// TIA Portal V20 export
ORGANIZATION_BLOCK "Startup"   // OB100, LAD, Startup
TITLE = "Complete Restart"
// stored: AutoNumber false, IsIECCheckEnabled true, SetENOAutomatically true
   VAR_INPUT
      LostRetentive : Bool;   // True if retentive data are lost
      LostRTC : Bool;   // True if date and time are lost
   END_VAR
   VAR_TEMP
      tempError : Bool;
      tempStatus : Word;
      tempDiagnostics : "LAF_typeDiagnosticsSimple";
   END_VAR
BEGIN

REGION Network 1: Erster Zyklus bit setzen / Set first cycle bit
   // Setze das "erster Zyklus" Signal und die Signale immer EIN sowie immer AUS / Set the first cycle signal
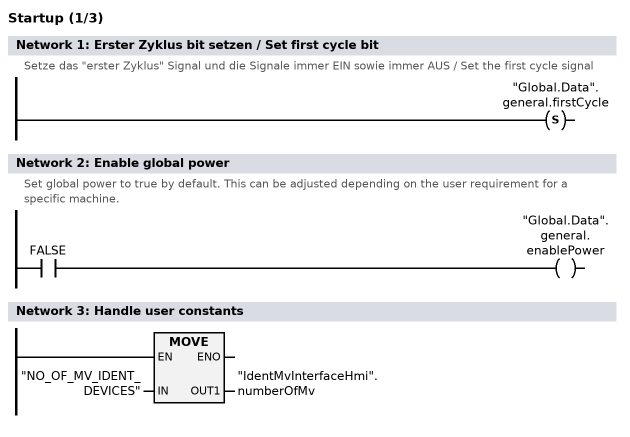
   RUNG wire#powerrail
      S_Coil( "Global.Data".general.firstCycle )
   END_RUNG
   // the same network as SCL:
   "Global.Data".general.firstCycle := TRUE;
END_REGION

REGION Network 2: Enable global power
   // Set global power to true by default. This can be adjusted depending on the user requirement for a specific machine.
   RUNG wire#powerrail
      Contact( FALSE )
      Coil( "Global.Data".general.enablePower )
   END_RUNG
   // the same network as SCL:
   "Global.Data".general.enablePower := FALSE;
END_REGION

REGION Network 3: Handle user constants
   RUNG wire#powerrail
      Move(in := "NO_OF_MV_IDENT_DEVICES", out1 => "IdentMvInterfaceHmi".numberOfMv)
   END_RUNG
   // the same network as SCL:
   "IdentMvInterfaceHmi".numberOfMv := "NO_OF_MV_IDENT_DEVICES";
END_REGION

REGION Network 4: Set drive objects for drive diagnostic
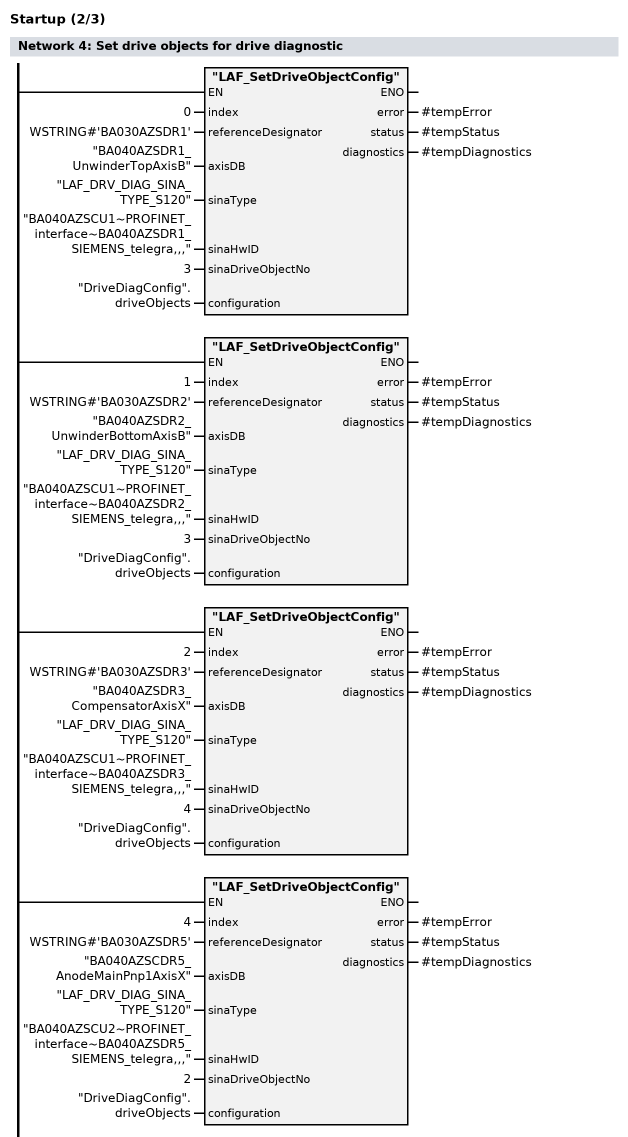
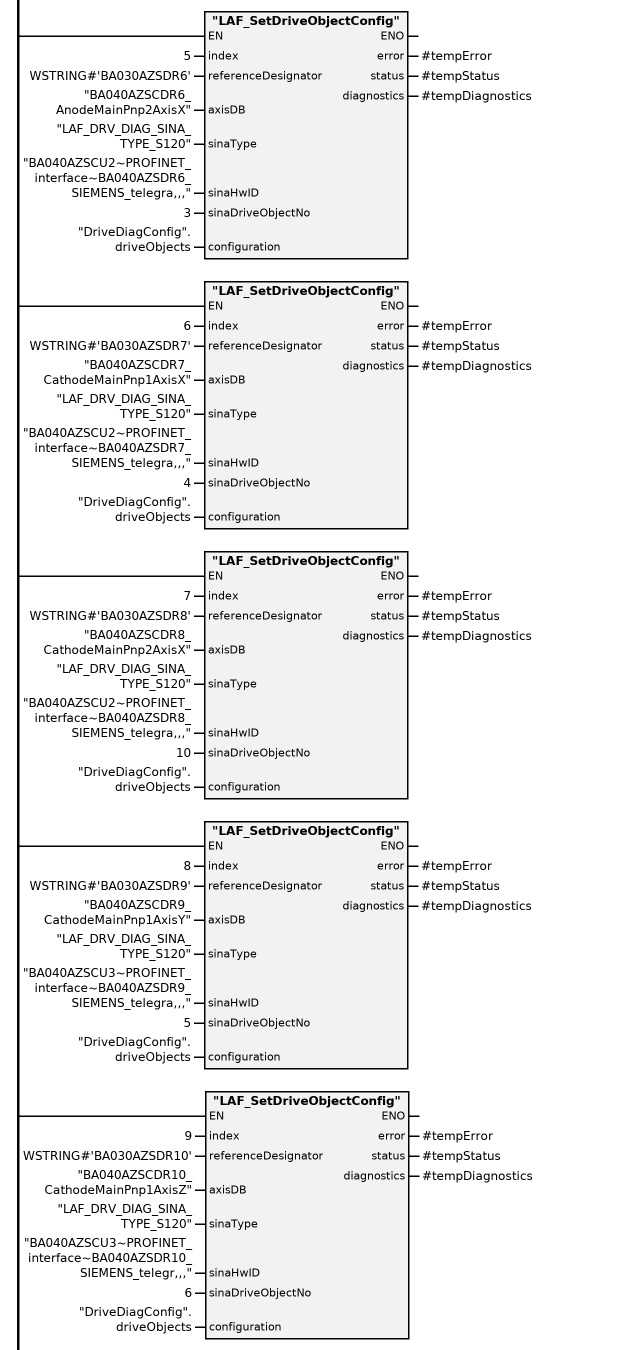
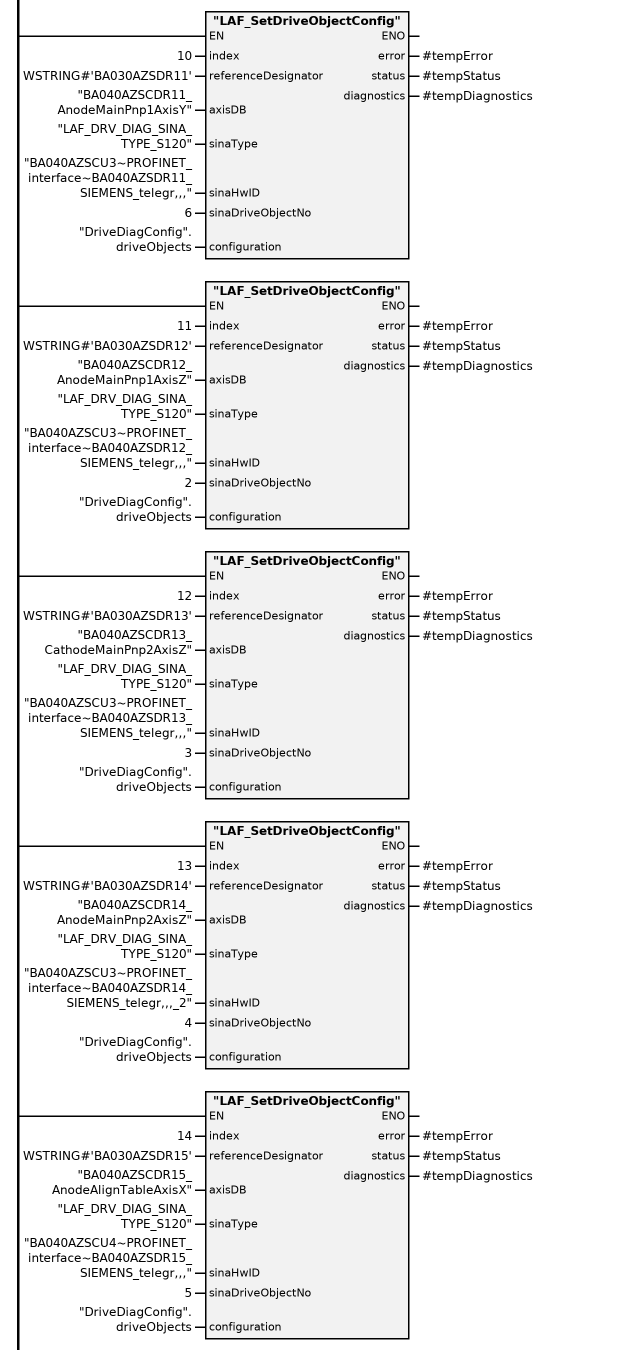
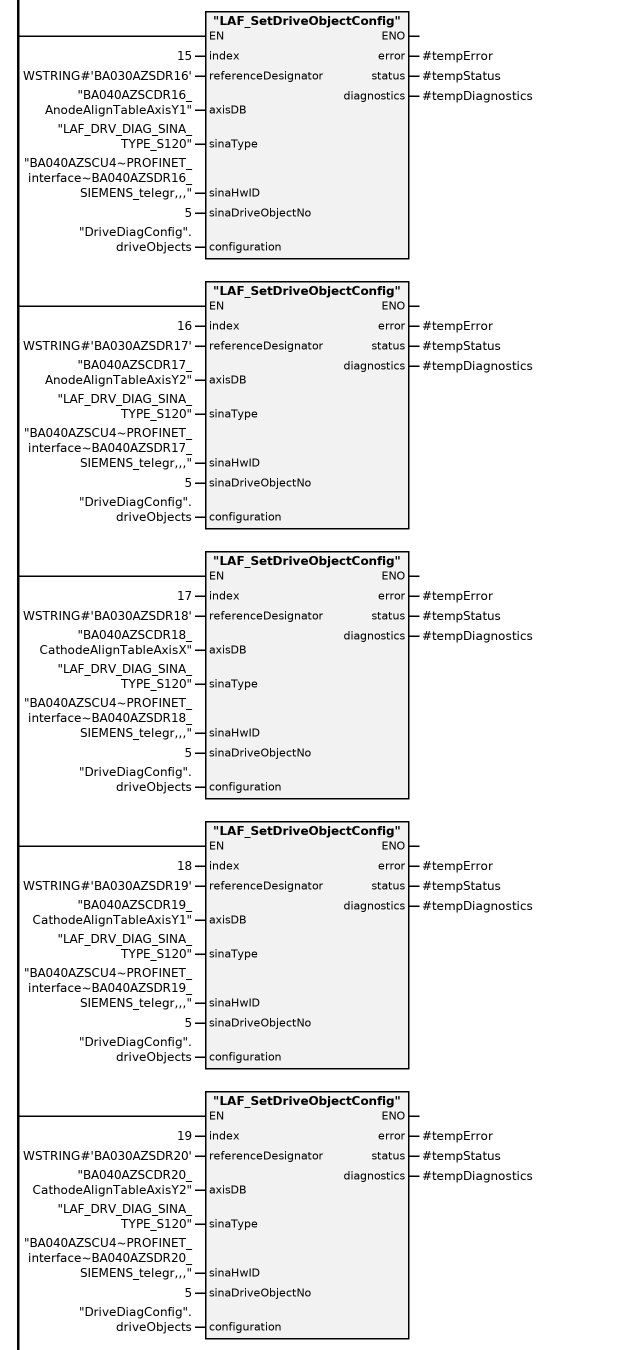
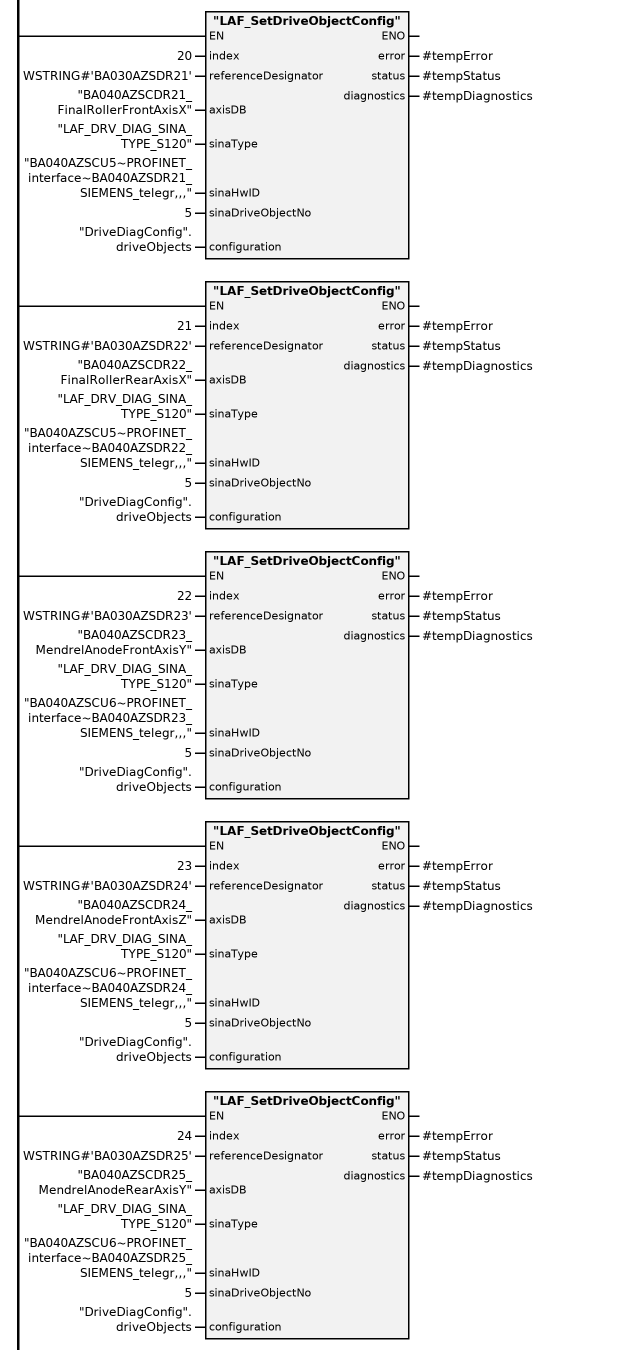
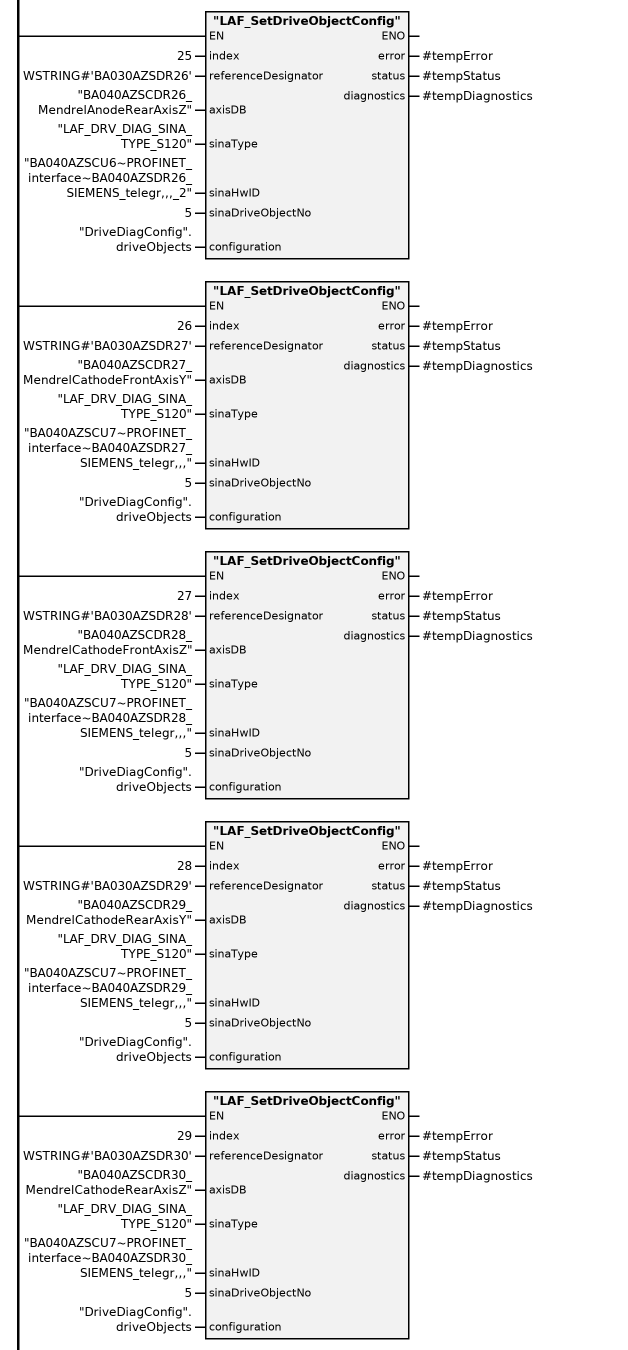
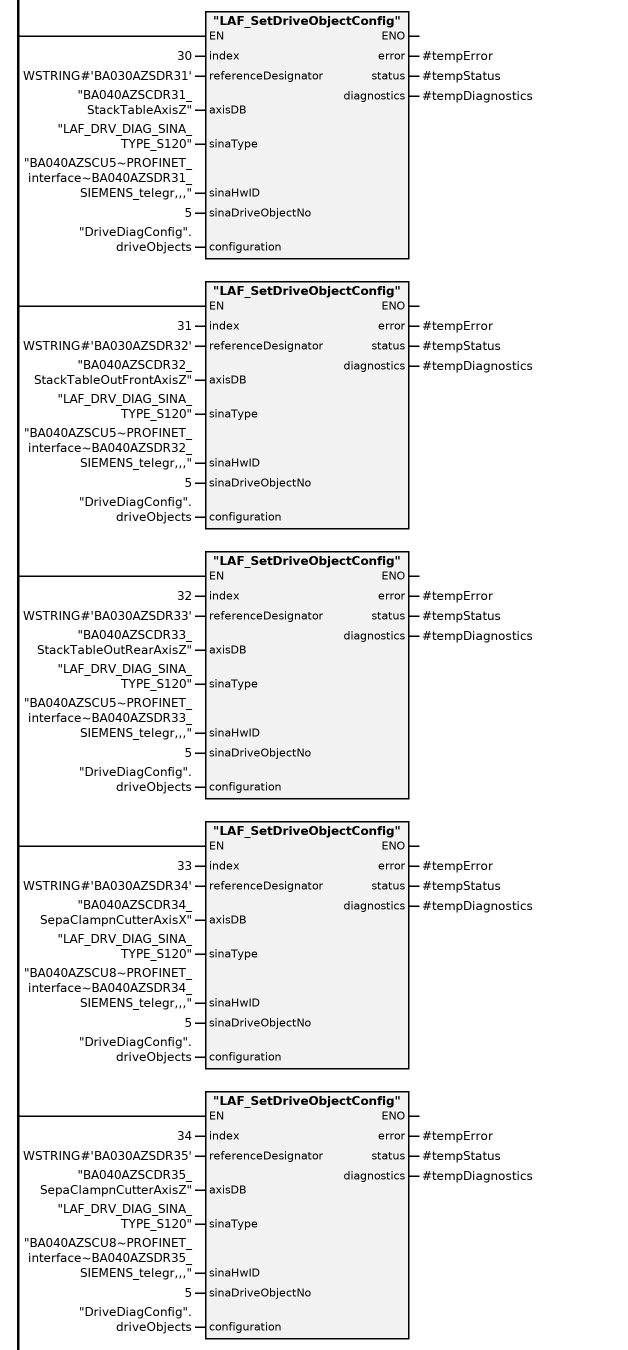
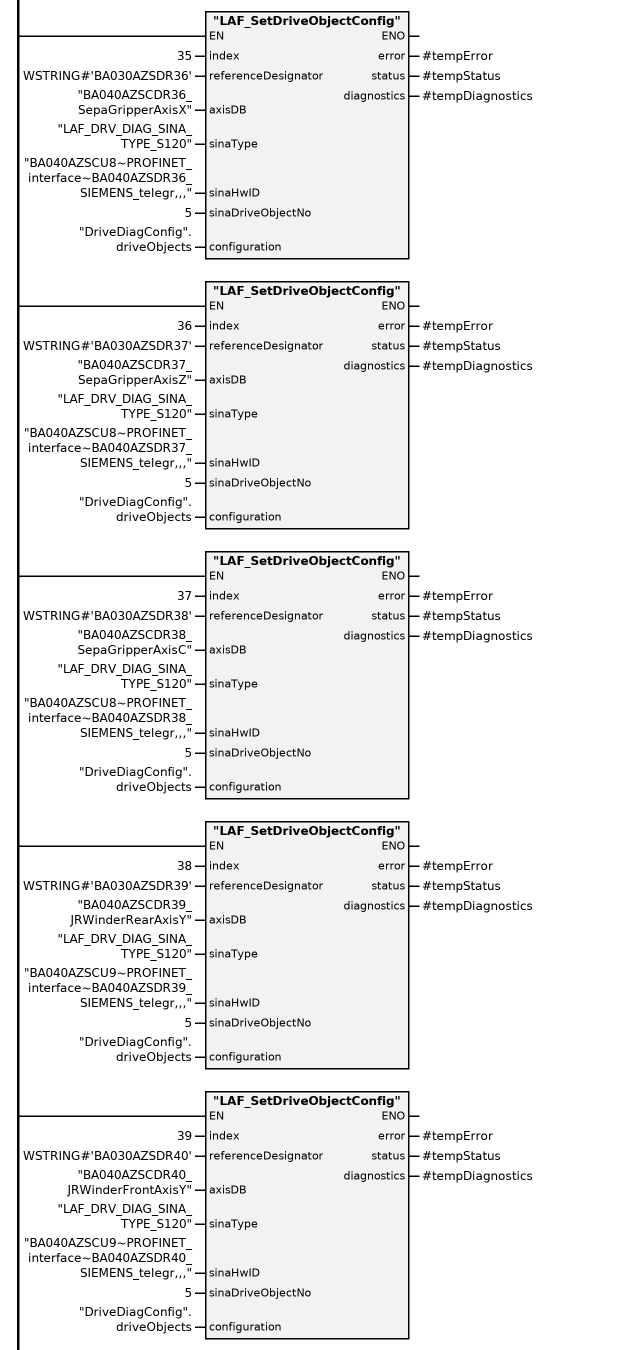
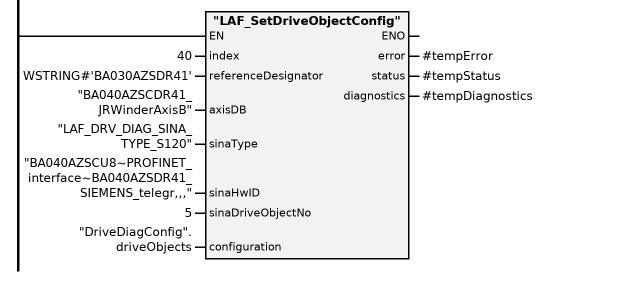
   RUNG wire#powerrail
      "LAF_SetDriveObjectConfig"(index := 0, referenceDesignator := WSTRING#'BA030AZSDR1', axisDB := "BA040AZSDR1_UnwinderTopAxisB", sinaType := "LAF_DRV_DIAG_SINA_TYPE_S120", sinaHwID := "BA040AZSCU1~PROFINET_interface~BA040AZSDR1_SIEMENS_telegra,,,", sinaDriveObjectNo := 3, configuration := "DriveDiagConfig".driveObjects, error => #tempError, status => #tempStatus, diagnostics => #tempDiagnostics)
   END_RUNG
   RUNG wire#powerrail
      "LAF_SetDriveObjectConfig"(index := 1, referenceDesignator := WSTRING#'BA030AZSDR2', axisDB := "BA040AZSDR2_UnwinderBottomAxisB", sinaType := "LAF_DRV_DIAG_SINA_TYPE_S120", sinaHwID := "BA040AZSCU1~PROFINET_interface~BA040AZSDR2_SIEMENS_telegra,,,", sinaDriveObjectNo := 3, configuration := "DriveDiagConfig".driveObjects, error => #tempError, status => #tempStatus, diagnostics => #tempDiagnostics)
   END_RUNG
   RUNG wire#powerrail
      "LAF_SetDriveObjectConfig"(index := 2, referenceDesignator := WSTRING#'BA030AZSDR3', axisDB := "BA040AZSDR3_CompensatorAxisX", sinaType := "LAF_DRV_DIAG_SINA_TYPE_S120", sinaHwID := "BA040AZSCU1~PROFINET_interface~BA040AZSDR3_SIEMENS_telegra,,,", sinaDriveObjectNo := 4, configuration := "DriveDiagConfig".driveObjects, error => #tempError, status => #tempStatus, diagnostics => #tempDiagnostics)
   END_RUNG
   RUNG wire#powerrail
      "LAF_SetDriveObjectConfig"(index := 4, referenceDesignator := WSTRING#'BA030AZSDR5', axisDB := "BA040AZSCDR5_AnodeMainPnp1AxisX", sinaType := "LAF_DRV_DIAG_SINA_TYPE_S120", sinaHwID := "BA040AZSCU2~PROFINET_interface~BA040AZSDR5_SIEMENS_telegra,,,", sinaDriveObjectNo := 2, configuration := "DriveDiagConfig".driveObjects, error => #tempError, status => #tempStatus, diagnostics => #tempDiagnostics)
   END_RUNG
   RUNG wire#powerrail
      "LAF_SetDriveObjectConfig"(index := 5, referenceDesignator := WSTRING#'BA030AZSDR6', axisDB := "BA040AZSCDR6_AnodeMainPnp2AxisX", sinaType := "LAF_DRV_DIAG_SINA_TYPE_S120", sinaHwID := "BA040AZSCU2~PROFINET_interface~BA040AZSDR6_SIEMENS_telegra,,,", sinaDriveObjectNo := 3, configuration := "DriveDiagConfig".driveObjects, error => #tempError, status => #tempStatus, diagnostics => #tempDiagnostics)
   END_RUNG
   RUNG wire#powerrail
      "LAF_SetDriveObjectConfig"(index := 6, referenceDesignator := WSTRING#'BA030AZSDR7', axisDB := "BA040AZSCDR7_CathodeMainPnp1AxisX", sinaType := "LAF_DRV_DIAG_SINA_TYPE_S120", sinaHwID := "BA040AZSCU2~PROFINET_interface~BA040AZSDR7_SIEMENS_telegra,,,", sinaDriveObjectNo := 4, configuration := "DriveDiagConfig".driveObjects, error => #tempError, status => #tempStatus, diagnostics => #tempDiagnostics)
   END_RUNG
   RUNG wire#powerrail
      "LAF_SetDriveObjectConfig"(index := 7, referenceDesignator := WSTRING#'BA030AZSDR8', axisDB := "BA040AZSCDR8_CathodeMainPnp2AxisX", sinaType := "LAF_DRV_DIAG_SINA_TYPE_S120", sinaHwID := "BA040AZSCU2~PROFINET_interface~BA040AZSDR8_SIEMENS_telegra,,,", sinaDriveObjectNo := 10, configuration := "DriveDiagConfig".driveObjects, error => #tempError, status => #tempStatus, diagnostics => #tempDiagnostics)
   END_RUNG
   RUNG wire#powerrail
      "LAF_SetDriveObjectConfig"(index := 8, referenceDesignator := WSTRING#'BA030AZSDR9', axisDB := "BA040AZSCDR9_CathodeMainPnp1AxisY", sinaType := "LAF_DRV_DIAG_SINA_TYPE_S120", sinaHwID := "BA040AZSCU3~PROFINET_interface~BA040AZSDR9_SIEMENS_telegra,,,", sinaDriveObjectNo := 5, configuration := "DriveDiagConfig".driveObjects, error => #tempError, status => #tempStatus, diagnostics => #tempDiagnostics)
   END_RUNG
   RUNG wire#powerrail
      "LAF_SetDriveObjectConfig"(index := 9, referenceDesignator := WSTRING#'BA030AZSDR10', axisDB := "BA040AZSCDR10_CathodeMainPnp1AxisZ", sinaType := "LAF_DRV_DIAG_SINA_TYPE_S120", sinaHwID := "BA040AZSCU3~PROFINET_interface~BA040AZSDR10_SIEMENS_telegr,,,", sinaDriveObjectNo := 6, configuration := "DriveDiagConfig".driveObjects, error => #tempError, status => #tempStatus, diagnostics => #tempDiagnostics)
   END_RUNG
   RUNG wire#powerrail
      "LAF_SetDriveObjectConfig"(index := 10, referenceDesignator := WSTRING#'BA030AZSDR11', axisDB := "BA040AZSCDR11_AnodeMainPnp1AxisY", sinaType := "LAF_DRV_DIAG_SINA_TYPE_S120", sinaHwID := "BA040AZSCU3~PROFINET_interface~BA040AZSDR11_SIEMENS_telegr,,,", sinaDriveObjectNo := 6, configuration := "DriveDiagConfig".driveObjects, error => #tempError, status => #tempStatus, diagnostics => #tempDiagnostics)
   END_RUNG
   RUNG wire#powerrail
      "LAF_SetDriveObjectConfig"(index := 11, referenceDesignator := WSTRING#'BA030AZSDR12', axisDB := "BA040AZSCDR12_AnodeMainPnp1AxisZ", sinaType := "LAF_DRV_DIAG_SINA_TYPE_S120", sinaHwID := "BA040AZSCU3~PROFINET_interface~BA040AZSDR12_SIEMENS_telegr,,,", sinaDriveObjectNo := 2, configuration := "DriveDiagConfig".driveObjects, error => #tempError, status => #tempStatus, diagnostics => #tempDiagnostics)
   END_RUNG
   RUNG wire#powerrail
      "LAF_SetDriveObjectConfig"(index := 12, referenceDesignator := WSTRING#'BA030AZSDR13', axisDB := "BA040AZSCDR13_CathodeMainPnp2AxisZ", sinaType := "LAF_DRV_DIAG_SINA_TYPE_S120", sinaHwID := "BA040AZSCU3~PROFINET_interface~BA040AZSDR13_SIEMENS_telegr,,,", sinaDriveObjectNo := 3, configuration := "DriveDiagConfig".driveObjects, error => #tempError, status => #tempStatus, diagnostics => #tempDiagnostics)
   END_RUNG
   RUNG wire#powerrail
      "LAF_SetDriveObjectConfig"(index := 13, referenceDesignator := WSTRING#'BA030AZSDR14', axisDB := "BA040AZSCDR14_AnodeMainPnp2AxisZ", sinaType := "LAF_DRV_DIAG_SINA_TYPE_S120", sinaHwID := "BA040AZSCU3~PROFINET_interface~BA040AZSDR14_SIEMENS_telegr,,,_2", sinaDriveObjectNo := 4, configuration := "DriveDiagConfig".driveObjects, error => #tempError, status => #tempStatus, diagnostics => #tempDiagnostics)
   END_RUNG
   RUNG wire#powerrail
      "LAF_SetDriveObjectConfig"(index := 14, referenceDesignator := WSTRING#'BA030AZSDR15', axisDB := "BA040AZSCDR15_AnodeAlignTableAxisX", sinaType := "LAF_DRV_DIAG_SINA_TYPE_S120", sinaHwID := "BA040AZSCU4~PROFINET_interface~BA040AZSDR15_SIEMENS_telegr,,,", sinaDriveObjectNo := 5, configuration := "DriveDiagConfig".driveObjects, error => #tempError, status => #tempStatus, diagnostics => #tempDiagnostics)
   END_RUNG
   RUNG wire#powerrail
      "LAF_SetDriveObjectConfig"(index := 15, referenceDesignator := WSTRING#'BA030AZSDR16', axisDB := "BA040AZSCDR16_AnodeAlignTableAxisY1", sinaType := "LAF_DRV_DIAG_SINA_TYPE_S120", sinaHwID := "BA040AZSCU4~PROFINET_interface~BA040AZSDR16_SIEMENS_telegr,,,", sinaDriveObjectNo := 5, configuration := "DriveDiagConfig".driveObjects, error => #tempError, status => #tempStatus, diagnostics => #tempDiagnostics)
   END_RUNG
   RUNG wire#powerrail
      "LAF_SetDriveObjectConfig"(index := 16, referenceDesignator := WSTRING#'BA030AZSDR17', axisDB := "BA040AZSCDR17_AnodeAlignTableAxisY2", sinaType := "LAF_DRV_DIAG_SINA_TYPE_S120", sinaHwID := "BA040AZSCU4~PROFINET_interface~BA040AZSDR17_SIEMENS_telegr,,,", sinaDriveObjectNo := 5, configuration := "DriveDiagConfig".driveObjects, error => #tempError, status => #tempStatus, diagnostics => #tempDiagnostics)
   END_RUNG
   RUNG wire#powerrail
      "LAF_SetDriveObjectConfig"(index := 17, referenceDesignator := WSTRING#'BA030AZSDR18', axisDB := "BA040AZSCDR18_CathodeAlignTableAxisX", sinaType := "LAF_DRV_DIAG_SINA_TYPE_S120", sinaHwID := "BA040AZSCU4~PROFINET_interface~BA040AZSDR18_SIEMENS_telegr,,,", sinaDriveObjectNo := 5, configuration := "DriveDiagConfig".driveObjects, error => #tempError, status => #tempStatus, diagnostics => #tempDiagnostics)
   END_RUNG
   RUNG wire#powerrail
      "LAF_SetDriveObjectConfig"(index := 18, referenceDesignator := WSTRING#'BA030AZSDR19', axisDB := "BA040AZSCDR19_CathodeAlignTableAxisY1", sinaType := "LAF_DRV_DIAG_SINA_TYPE_S120", sinaHwID := "BA040AZSCU4~PROFINET_interface~BA040AZSDR19_SIEMENS_telegr,,,", sinaDriveObjectNo := 5, configuration := "DriveDiagConfig".driveObjects, error => #tempError, status => #tempStatus, diagnostics => #tempDiagnostics)
   END_RUNG
   RUNG wire#powerrail
      "LAF_SetDriveObjectConfig"(index := 19, referenceDesignator := WSTRING#'BA030AZSDR20', axisDB := "BA040AZSCDR20_CathodeAlignTableAxisY2", sinaType := "LAF_DRV_DIAG_SINA_TYPE_S120", sinaHwID := "BA040AZSCU4~PROFINET_interface~BA040AZSDR20_SIEMENS_telegr,,,", sinaDriveObjectNo := 5, configuration := "DriveDiagConfig".driveObjects, error => #tempError, status => #tempStatus, diagnostics => #tempDiagnostics)
   END_RUNG
   RUNG wire#powerrail
      "LAF_SetDriveObjectConfig"(index := 20, referenceDesignator := WSTRING#'BA030AZSDR21', axisDB := "BA040AZSCDR21_FinalRollerFrontAxisX", sinaType := "LAF_DRV_DIAG_SINA_TYPE_S120", sinaHwID := "BA040AZSCU5~PROFINET_interface~BA040AZSDR21_SIEMENS_telegr,,,", sinaDriveObjectNo := 5, configuration := "DriveDiagConfig".driveObjects, error => #tempError, status => #tempStatus, diagnostics => #tempDiagnostics)
   END_RUNG
   RUNG wire#powerrail
      "LAF_SetDriveObjectConfig"(index := 21, referenceDesignator := WSTRING#'BA030AZSDR22', axisDB := "BA040AZSCDR22_FinalRollerRearAxisX", sinaType := "LAF_DRV_DIAG_SINA_TYPE_S120", sinaHwID := "BA040AZSCU5~PROFINET_interface~BA040AZSDR22_SIEMENS_telegr,,,", sinaDriveObjectNo := 5, configuration := "DriveDiagConfig".driveObjects, error => #tempError, status => #tempStatus, diagnostics => #tempDiagnostics)
   END_RUNG
   RUNG wire#powerrail
      "LAF_SetDriveObjectConfig"(index := 22, referenceDesignator := WSTRING#'BA030AZSDR23', axisDB := "BA040AZSCDR23_MendrelAnodeFrontAxisY", sinaType := "LAF_DRV_DIAG_SINA_TYPE_S120", sinaHwID := "BA040AZSCU6~PROFINET_interface~BA040AZSDR23_SIEMENS_telegr,,,", sinaDriveObjectNo := 5, configuration := "DriveDiagConfig".driveObjects, error => #tempError, status => #tempStatus, diagnostics => #tempDiagnostics)
   END_RUNG
   RUNG wire#powerrail
      "LAF_SetDriveObjectConfig"(index := 23, referenceDesignator := WSTRING#'BA030AZSDR24', axisDB := "BA040AZSCDR24_MendrelAnodeFrontAxisZ", sinaType := "LAF_DRV_DIAG_SINA_TYPE_S120", sinaHwID := "BA040AZSCU6~PROFINET_interface~BA040AZSDR24_SIEMENS_telegr,,,", sinaDriveObjectNo := 5, configuration := "DriveDiagConfig".driveObjects, error => #tempError, status => #tempStatus, diagnostics => #tempDiagnostics)
   END_RUNG
   RUNG wire#powerrail
      "LAF_SetDriveObjectConfig"(index := 24, referenceDesignator := WSTRING#'BA030AZSDR25', axisDB := "BA040AZSCDR25_MendrelAnodeRearAxisY", sinaType := "LAF_DRV_DIAG_SINA_TYPE_S120", sinaHwID := "BA040AZSCU6~PROFINET_interface~BA040AZSDR25_SIEMENS_telegr,,,", sinaDriveObjectNo := 5, configuration := "DriveDiagConfig".driveObjects, error => #tempError, status => #tempStatus, diagnostics => #tempDiagnostics)
   END_RUNG
   RUNG wire#powerrail
      "LAF_SetDriveObjectConfig"(index := 25, referenceDesignator := WSTRING#'BA030AZSDR26', axisDB := "BA040AZSCDR26_MendrelAnodeRearAxisZ", sinaType := "LAF_DRV_DIAG_SINA_TYPE_S120", sinaHwID := "BA040AZSCU6~PROFINET_interface~BA040AZSDR26_SIEMENS_telegr,,,_2", sinaDriveObjectNo := 5, configuration := "DriveDiagConfig".driveObjects, error => #tempError, status => #tempStatus, diagnostics => #tempDiagnostics)
   END_RUNG
   RUNG wire#powerrail
      "LAF_SetDriveObjectConfig"(index := 26, referenceDesignator := WSTRING#'BA030AZSDR27', axisDB := "BA040AZSCDR27_MendrelCathodeFrontAxisY", sinaType := "LAF_DRV_DIAG_SINA_TYPE_S120", sinaHwID := "BA040AZSCU7~PROFINET_interface~BA040AZSDR27_SIEMENS_telegr,,,", sinaDriveObjectNo := 5, configuration := "DriveDiagConfig".driveObjects, error => #tempError, status => #tempStatus, diagnostics => #tempDiagnostics)
   END_RUNG
   RUNG wire#powerrail
      "LAF_SetDriveObjectConfig"(index := 27, referenceDesignator := WSTRING#'BA030AZSDR28', axisDB := "BA040AZSCDR28_MendrelCathodeFrontAxisZ", sinaType := "LAF_DRV_DIAG_SINA_TYPE_S120", sinaHwID := "BA040AZSCU7~PROFINET_interface~BA040AZSDR28_SIEMENS_telegr,,,", sinaDriveObjectNo := 5, configuration := "DriveDiagConfig".driveObjects, error => #tempError, status => #tempStatus, diagnostics => #tempDiagnostics)
   END_RUNG
   RUNG wire#powerrail
      "LAF_SetDriveObjectConfig"(index := 28, referenceDesignator := WSTRING#'BA030AZSDR29', axisDB := "BA040AZSCDR29_MendrelCathodeRearAxisY", sinaType := "LAF_DRV_DIAG_SINA_TYPE_S120", sinaHwID := "BA040AZSCU7~PROFINET_interface~BA040AZSDR29_SIEMENS_telegr,,,", sinaDriveObjectNo := 5, configuration := "DriveDiagConfig".driveObjects, error => #tempError, status => #tempStatus, diagnostics => #tempDiagnostics)
   END_RUNG
   RUNG wire#powerrail
      "LAF_SetDriveObjectConfig"(index := 29, referenceDesignator := WSTRING#'BA030AZSDR30', axisDB := "BA040AZSCDR30_MendrelCathodeRearAxisZ", sinaType := "LAF_DRV_DIAG_SINA_TYPE_S120", sinaHwID := "BA040AZSCU7~PROFINET_interface~BA040AZSDR30_SIEMENS_telegr,,,", sinaDriveObjectNo := 5, configuration := "DriveDiagConfig".driveObjects, error => #tempError, status => #tempStatus, diagnostics => #tempDiagnostics)
   END_RUNG
   RUNG wire#powerrail
      "LAF_SetDriveObjectConfig"(index := 30, referenceDesignator := WSTRING#'BA030AZSDR31', axisDB := "BA040AZSCDR31_StackTableAxisZ", sinaType := "LAF_DRV_DIAG_SINA_TYPE_S120", sinaHwID := "BA040AZSCU5~PROFINET_interface~BA040AZSDR31_SIEMENS_telegr,,,", sinaDriveObjectNo := 5, configuration := "DriveDiagConfig".driveObjects, error => #tempError, status => #tempStatus, diagnostics => #tempDiagnostics)
   END_RUNG
   RUNG wire#powerrail
      "LAF_SetDriveObjectConfig"(index := 31, referenceDesignator := WSTRING#'BA030AZSDR32', axisDB := "BA040AZSCDR32_StackTableOutFrontAxisZ", sinaType := "LAF_DRV_DIAG_SINA_TYPE_S120", sinaHwID := "BA040AZSCU5~PROFINET_interface~BA040AZSDR32_SIEMENS_telegr,,,", sinaDriveObjectNo := 5, configuration := "DriveDiagConfig".driveObjects, error => #tempError, status => #tempStatus, diagnostics => #tempDiagnostics)
   END_RUNG
   RUNG wire#powerrail
      "LAF_SetDriveObjectConfig"(index := 32, referenceDesignator := WSTRING#'BA030AZSDR33', axisDB := "BA040AZSCDR33_StackTableOutRearAxisZ", sinaType := "LAF_DRV_DIAG_SINA_TYPE_S120", sinaHwID := "BA040AZSCU5~PROFINET_interface~BA040AZSDR33_SIEMENS_telegr,,,", sinaDriveObjectNo := 5, configuration := "DriveDiagConfig".driveObjects, error => #tempError, status => #tempStatus, diagnostics => #tempDiagnostics)
   END_RUNG
   RUNG wire#powerrail
      "LAF_SetDriveObjectConfig"(index := 33, referenceDesignator := WSTRING#'BA030AZSDR34', axisDB := "BA040AZSCDR34_SepaClampnCutterAxisX", sinaType := "LAF_DRV_DIAG_SINA_TYPE_S120", sinaHwID := "BA040AZSCU8~PROFINET_interface~BA040AZSDR34_SIEMENS_telegr,,,", sinaDriveObjectNo := 5, configuration := "DriveDiagConfig".driveObjects, error => #tempError, status => #tempStatus, diagnostics => #tempDiagnostics)
   END_RUNG
   RUNG wire#powerrail
      "LAF_SetDriveObjectConfig"(index := 34, referenceDesignator := WSTRING#'BA030AZSDR35', axisDB := "BA040AZSCDR35_SepaClampnCutterAxisZ", sinaType := "LAF_DRV_DIAG_SINA_TYPE_S120", sinaHwID := "BA040AZSCU8~PROFINET_interface~BA040AZSDR35_SIEMENS_telegr,,,", sinaDriveObjectNo := 5, configuration := "DriveDiagConfig".driveObjects, error => #tempError, status => #tempStatus, diagnostics => #tempDiagnostics)
   END_RUNG
   RUNG wire#powerrail
      "LAF_SetDriveObjectConfig"(index := 35, referenceDesignator := WSTRING#'BA030AZSDR36', axisDB := "BA040AZSCDR36_SepaGripperAxisX", sinaType := "LAF_DRV_DIAG_SINA_TYPE_S120", sinaHwID := "BA040AZSCU8~PROFINET_interface~BA040AZSDR36_SIEMENS_telegr,,,", sinaDriveObjectNo := 5, configuration := "DriveDiagConfig".driveObjects, error => #tempError, status => #tempStatus, diagnostics => #tempDiagnostics)
   END_RUNG
   RUNG wire#powerrail
      "LAF_SetDriveObjectConfig"(index := 36, referenceDesignator := WSTRING#'BA030AZSDR37', axisDB := "BA040AZSCDR37_SepaGripperAxisZ", sinaType := "LAF_DRV_DIAG_SINA_TYPE_S120", sinaHwID := "BA040AZSCU8~PROFINET_interface~BA040AZSDR37_SIEMENS_telegr,,,", sinaDriveObjectNo := 5, configuration := "DriveDiagConfig".driveObjects, error => #tempError, status => #tempStatus, diagnostics => #tempDiagnostics)
   END_RUNG
   RUNG wire#powerrail
      "LAF_SetDriveObjectConfig"(index := 37, referenceDesignator := WSTRING#'BA030AZSDR38', axisDB := "BA040AZSCDR38_SepaGripperAxisC", sinaType := "LAF_DRV_DIAG_SINA_TYPE_S120", sinaHwID := "BA040AZSCU8~PROFINET_interface~BA040AZSDR38_SIEMENS_telegr,,,", sinaDriveObjectNo := 5, configuration := "DriveDiagConfig".driveObjects, error => #tempError, status => #tempStatus, diagnostics => #tempDiagnostics)
   END_RUNG
   RUNG wire#powerrail
      "LAF_SetDriveObjectConfig"(index := 38, referenceDesignator := WSTRING#'BA030AZSDR39', axisDB := "BA040AZSCDR39_JRWinderRearAxisY", sinaType := "LAF_DRV_DIAG_SINA_TYPE_S120", sinaHwID := "BA040AZSCU9~PROFINET_interface~BA040AZSDR39_SIEMENS_telegr,,,", sinaDriveObjectNo := 5, configuration := "DriveDiagConfig".driveObjects, error => #tempError, status => #tempStatus, diagnostics => #tempDiagnostics)
   END_RUNG
   RUNG wire#powerrail
      "LAF_SetDriveObjectConfig"(index := 39, referenceDesignator := WSTRING#'BA030AZSDR40', axisDB := "BA040AZSCDR40_JRWinderFrontAxisY", sinaType := "LAF_DRV_DIAG_SINA_TYPE_S120", sinaHwID := "BA040AZSCU9~PROFINET_interface~BA040AZSDR40_SIEMENS_telegr,,,", sinaDriveObjectNo := 5, configuration := "DriveDiagConfig".driveObjects, error => #tempError, status => #tempStatus, diagnostics => #tempDiagnostics)
   END_RUNG
   RUNG wire#powerrail
      "LAF_SetDriveObjectConfig"(index := 40, referenceDesignator := WSTRING#'BA030AZSDR41', axisDB := "BA040AZSCDR41_JRWinderAxisB", sinaType := "LAF_DRV_DIAG_SINA_TYPE_S120", sinaHwID := "BA040AZSCU8~PROFINET_interface~BA040AZSDR41_SIEMENS_telegr,,,", sinaDriveObjectNo := 5, configuration := "DriveDiagConfig".driveObjects, error => #tempError, status => #tempStatus, diagnostics => #tempDiagnostics)
   END_RUNG
   // the same network as SCL:
   "LAF_SetDriveObjectConfig"(index := 0,
                           referenceDesignator := WSTRING#'BA030AZSDR1',
                           axisDB := "BA040AZSDR1_UnwinderTopAxisB",
                           sinaType := "LAF_DRV_DIAG_SINA_TYPE_S120",
                           sinaHwID := "BA040AZSCU1~PROFINET_interface~BA040AZSDR1_SIEMENS_telegra,,,",
                           sinaDriveObjectNo := 3,
                           configuration := "DriveDiagConfig".driveObjects,
                           error => #tempError,
                           status => #tempStatus,
                           diagnostics => #tempDiagnostics);
   "LAF_SetDriveObjectConfig"(index := 1,
                           referenceDesignator := WSTRING#'BA030AZSDR2',
                           axisDB := "BA040AZSDR2_UnwinderBottomAxisB",
                           sinaType := "LAF_DRV_DIAG_SINA_TYPE_S120",
                           sinaHwID := "BA040AZSCU1~PROFINET_interface~BA040AZSDR2_SIEMENS_telegra,,,",
                           sinaDriveObjectNo := 3,
                           configuration := "DriveDiagConfig".driveObjects,
                           error => #tempError,
                           status => #tempStatus,
                           diagnostics => #tempDiagnostics);
   "LAF_SetDriveObjectConfig"(index := 2,
                           referenceDesignator := WSTRING#'BA030AZSDR3',
                           axisDB := "BA040AZSDR3_CompensatorAxisX",
                           sinaType := "LAF_DRV_DIAG_SINA_TYPE_S120",
                           sinaHwID := "BA040AZSCU1~PROFINET_interface~BA040AZSDR3_SIEMENS_telegra,,,",
                           sinaDriveObjectNo := 4,
                           configuration := "DriveDiagConfig".driveObjects,
                           error => #tempError,
                           status => #tempStatus,
                           diagnostics => #tempDiagnostics);
   "LAF_SetDriveObjectConfig"(index := 4,
                           referenceDesignator := WSTRING#'BA030AZSDR5',
                           axisDB := "BA040AZSCDR5_AnodeMainPnp1AxisX",
                           sinaType := "LAF_DRV_DIAG_SINA_TYPE_S120",
                           sinaHwID := "BA040AZSCU2~PROFINET_interface~BA040AZSDR5_SIEMENS_telegra,,,",
                           sinaDriveObjectNo := 2,
                           configuration := "DriveDiagConfig".driveObjects,
                           error => #tempError,
                           status => #tempStatus,
                           diagnostics => #tempDiagnostics);
   "LAF_SetDriveObjectConfig"(index := 5,
                           referenceDesignator := WSTRING#'BA030AZSDR6',
                           axisDB := "BA040AZSCDR6_AnodeMainPnp2AxisX",
                           sinaType := "LAF_DRV_DIAG_SINA_TYPE_S120",
                           sinaHwID := "BA040AZSCU2~PROFINET_interface~BA040AZSDR6_SIEMENS_telegra,,,",
                           sinaDriveObjectNo := 3,
                           configuration := "DriveDiagConfig".driveObjects,
                           error => #tempError,
                           status => #tempStatus,
                           diagnostics => #tempDiagnostics);
   "LAF_SetDriveObjectConfig"(index := 6,
                           referenceDesignator := WSTRING#'BA030AZSDR7',
                           axisDB := "BA040AZSCDR7_CathodeMainPnp1AxisX",
                           sinaType := "LAF_DRV_DIAG_SINA_TYPE_S120",
                           sinaHwID := "BA040AZSCU2~PROFINET_interface~BA040AZSDR7_SIEMENS_telegra,,,",
                           sinaDriveObjectNo := 4,
                           configuration := "DriveDiagConfig".driveObjects,
                           error => #tempError,
                           status => #tempStatus,
                           diagnostics => #tempDiagnostics);
   "LAF_SetDriveObjectConfig"(index := 7,
                           referenceDesignator := WSTRING#'BA030AZSDR8',
                           axisDB := "BA040AZSCDR8_CathodeMainPnp2AxisX",
                           sinaType := "LAF_DRV_DIAG_SINA_TYPE_S120",
                           sinaHwID := "BA040AZSCU2~PROFINET_interface~BA040AZSDR8_SIEMENS_telegra,,,",
                           sinaDriveObjectNo := 10,
                           configuration := "DriveDiagConfig".driveObjects,
                           error => #tempError,
                           status => #tempStatus,
                           diagnostics => #tempDiagnostics);
   "LAF_SetDriveObjectConfig"(index := 8,
                           referenceDesignator := WSTRING#'BA030AZSDR9',
                           axisDB := "BA040AZSCDR9_CathodeMainPnp1AxisY",
                           sinaType := "LAF_DRV_DIAG_SINA_TYPE_S120",
                           sinaHwID := "BA040AZSCU3~PROFINET_interface~BA040AZSDR9_SIEMENS_telegra,,,",
                           sinaDriveObjectNo := 5,
                           configuration := "DriveDiagConfig".driveObjects,
                           error => #tempError,
                           status => #tempStatus,
                           diagnostics => #tempDiagnostics);
   "LAF_SetDriveObjectConfig"(index := 9,
                           referenceDesignator := WSTRING#'BA030AZSDR10',
                           axisDB := "BA040AZSCDR10_CathodeMainPnp1AxisZ",
                           sinaType := "LAF_DRV_DIAG_SINA_TYPE_S120",
                           sinaHwID := "BA040AZSCU3~PROFINET_interface~BA040AZSDR10_SIEMENS_telegr,,,",
                           sinaDriveObjectNo := 6,
                           configuration := "DriveDiagConfig".driveObjects,
                           error => #tempError,
                           status => #tempStatus,
                           diagnostics => #tempDiagnostics);
   "LAF_SetDriveObjectConfig"(index := 10,
                           referenceDesignator := WSTRING#'BA030AZSDR11',
                           axisDB := "BA040AZSCDR11_AnodeMainPnp1AxisY",
                           sinaType := "LAF_DRV_DIAG_SINA_TYPE_S120",
                           sinaHwID := "BA040AZSCU3~PROFINET_interface~BA040AZSDR11_SIEMENS_telegr,,,",
                           sinaDriveObjectNo := 6,
                           configuration := "DriveDiagConfig".driveObjects,
                           error => #tempError,
                           status => #tempStatus,
                           diagnostics => #tempDiagnostics);
   "LAF_SetDriveObjectConfig"(index := 11,
                           referenceDesignator := WSTRING#'BA030AZSDR12',
                           axisDB := "BA040AZSCDR12_AnodeMainPnp1AxisZ",
                           sinaType := "LAF_DRV_DIAG_SINA_TYPE_S120",
                           sinaHwID := "BA040AZSCU3~PROFINET_interface~BA040AZSDR12_SIEMENS_telegr,,,",
                           sinaDriveObjectNo := 2,
                           configuration := "DriveDiagConfig".driveObjects,
                           error => #tempError,
                           status => #tempStatus,
                           diagnostics => #tempDiagnostics);
   "LAF_SetDriveObjectConfig"(index := 12,
                           referenceDesignator := WSTRING#'BA030AZSDR13',
                           axisDB := "BA040AZSCDR13_CathodeMainPnp2AxisZ",
                           sinaType := "LAF_DRV_DIAG_SINA_TYPE_S120",
                           sinaHwID := "BA040AZSCU3~PROFINET_interface~BA040AZSDR13_SIEMENS_telegr,,,",
                           sinaDriveObjectNo := 3,
                           configuration := "DriveDiagConfig".driveObjects,
                           error => #tempError,
                           status => #tempStatus,
                           diagnostics => #tempDiagnostics);
   "LAF_SetDriveObjectConfig"(index := 13,
                           referenceDesignator := WSTRING#'BA030AZSDR14',
                           axisDB := "BA040AZSCDR14_AnodeMainPnp2AxisZ",
                           sinaType := "LAF_DRV_DIAG_SINA_TYPE_S120",
                           sinaHwID := "BA040AZSCU3~PROFINET_interface~BA040AZSDR14_SIEMENS_telegr,,,_2",
                           sinaDriveObjectNo := 4,
                           configuration := "DriveDiagConfig".driveObjects,
                           error => #tempError,
                           status => #tempStatus,
                           diagnostics => #tempDiagnostics);
   "LAF_SetDriveObjectConfig"(index := 14,
                           referenceDesignator := WSTRING#'BA030AZSDR15',
                           axisDB := "BA040AZSCDR15_AnodeAlignTableAxisX",
                           sinaType := "LAF_DRV_DIAG_SINA_TYPE_S120",
                           sinaHwID := "BA040AZSCU4~PROFINET_interface~BA040AZSDR15_SIEMENS_telegr,,,",
                           sinaDriveObjectNo := 5,
                           configuration := "DriveDiagConfig".driveObjects,
                           error => #tempError,
                           status => #tempStatus,
                           diagnostics => #tempDiagnostics);
   "LAF_SetDriveObjectConfig"(index := 15,
                           referenceDesignator := WSTRING#'BA030AZSDR16',
                           axisDB := "BA040AZSCDR16_AnodeAlignTableAxisY1",
                           sinaType := "LAF_DRV_DIAG_SINA_TYPE_S120",
                           sinaHwID := "BA040AZSCU4~PROFINET_interface~BA040AZSDR16_SIEMENS_telegr,,,",
                           sinaDriveObjectNo := 5,
                           configuration := "DriveDiagConfig".driveObjects,
                           error => #tempError,
                           status => #tempStatus,
                           diagnostics => #tempDiagnostics);
   "LAF_SetDriveObjectConfig"(index := 16,
                           referenceDesignator := WSTRING#'BA030AZSDR17',
                           axisDB := "BA040AZSCDR17_AnodeAlignTableAxisY2",
                           sinaType := "LAF_DRV_DIAG_SINA_TYPE_S120",
                           sinaHwID := "BA040AZSCU4~PROFINET_interface~BA040AZSDR17_SIEMENS_telegr,,,",
                           sinaDriveObjectNo := 5,
                           configuration := "DriveDiagConfig".driveObjects,
                           error => #tempError,
                           status => #tempStatus,
                           diagnostics => #tempDiagnostics);
   "LAF_SetDriveObjectConfig"(index := 17,
                           referenceDesignator := WSTRING#'BA030AZSDR18',
                           axisDB := "BA040AZSCDR18_CathodeAlignTableAxisX",
                           sinaType := "LAF_DRV_DIAG_SINA_TYPE_S120",
                           sinaHwID := "BA040AZSCU4~PROFINET_interface~BA040AZSDR18_SIEMENS_telegr,,,",
                           sinaDriveObjectNo := 5,
                           configuration := "DriveDiagConfig".driveObjects,
                           error => #tempError,
                           status => #tempStatus,
                           diagnostics => #tempDiagnostics);
   "LAF_SetDriveObjectConfig"(index := 18,
                           referenceDesignator := WSTRING#'BA030AZSDR19',
                           axisDB := "BA040AZSCDR19_CathodeAlignTableAxisY1",
                           sinaType := "LAF_DRV_DIAG_SINA_TYPE_S120",
                           sinaHwID := "BA040AZSCU4~PROFINET_interface~BA040AZSDR19_SIEMENS_telegr,,,",
                           sinaDriveObjectNo := 5,
                           configuration := "DriveDiagConfig".driveObjects,
                           error => #tempError,
                           status => #tempStatus,
                           diagnostics => #tempDiagnostics);
   "LAF_SetDriveObjectConfig"(index := 19,
                           referenceDesignator := WSTRING#'BA030AZSDR20',
                           axisDB := "BA040AZSCDR20_CathodeAlignTableAxisY2",
                           sinaType := "LAF_DRV_DIAG_SINA_TYPE_S120",
                           sinaHwID := "BA040AZSCU4~PROFINET_interface~BA040AZSDR20_SIEMENS_telegr,,,",
                           sinaDriveObjectNo := 5,
                           configuration := "DriveDiagConfig".driveObjects,
                           error => #tempError,
                           status => #tempStatus,
                           diagnostics => #tempDiagnostics);
   "LAF_SetDriveObjectConfig"(index := 20,
                           referenceDesignator := WSTRING#'BA030AZSDR21',
                           axisDB := "BA040AZSCDR21_FinalRollerFrontAxisX",
                           sinaType := "LAF_DRV_DIAG_SINA_TYPE_S120",
                           sinaHwID := "BA040AZSCU5~PROFINET_interface~BA040AZSDR21_SIEMENS_telegr,,,",
                           sinaDriveObjectNo := 5,
                           configuration := "DriveDiagConfig".driveObjects,
                           error => #tempError,
                           status => #tempStatus,
                           diagnostics => #tempDiagnostics);
   "LAF_SetDriveObjectConfig"(index := 21,
                           referenceDesignator := WSTRING#'BA030AZSDR22',
                           axisDB := "BA040AZSCDR22_FinalRollerRearAxisX",
                           sinaType := "LAF_DRV_DIAG_SINA_TYPE_S120",
                           sinaHwID := "BA040AZSCU5~PROFINET_interface~BA040AZSDR22_SIEMENS_telegr,,,",
                           sinaDriveObjectNo := 5,
                           configuration := "DriveDiagConfig".driveObjects,
                           error => #tempError,
                           status => #tempStatus,
                           diagnostics => #tempDiagnostics);
   "LAF_SetDriveObjectConfig"(index := 22,
                           referenceDesignator := WSTRING#'BA030AZSDR23',
                           axisDB := "BA040AZSCDR23_MendrelAnodeFrontAxisY",
                           sinaType := "LAF_DRV_DIAG_SINA_TYPE_S120",
                           sinaHwID := "BA040AZSCU6~PROFINET_interface~BA040AZSDR23_SIEMENS_telegr,,,",
                           sinaDriveObjectNo := 5,
                           configuration := "DriveDiagConfig".driveObjects,
                           error => #tempError,
                           status => #tempStatus,
                           diagnostics => #tempDiagnostics);
   "LAF_SetDriveObjectConfig"(index := 23,
                           referenceDesignator := WSTRING#'BA030AZSDR24',
                           axisDB := "BA040AZSCDR24_MendrelAnodeFrontAxisZ",
                           sinaType := "LAF_DRV_DIAG_SINA_TYPE_S120",
                           sinaHwID := "BA040AZSCU6~PROFINET_interface~BA040AZSDR24_SIEMENS_telegr,,,",
                           sinaDriveObjectNo := 5,
                           configuration := "DriveDiagConfig".driveObjects,
                           error => #tempError,
                           status => #tempStatus,
                           diagnostics => #tempDiagnostics);
   "LAF_SetDriveObjectConfig"(index := 24,
                           referenceDesignator := WSTRING#'BA030AZSDR25',
                           axisDB := "BA040AZSCDR25_MendrelAnodeRearAxisY",
                           sinaType := "LAF_DRV_DIAG_SINA_TYPE_S120",
                           sinaHwID := "BA040AZSCU6~PROFINET_interface~BA040AZSDR25_SIEMENS_telegr,,,",
                           sinaDriveObjectNo := 5,
                           configuration := "DriveDiagConfig".driveObjects,
                           error => #tempError,
                           status => #tempStatus,
                           diagnostics => #tempDiagnostics);
   "LAF_SetDriveObjectConfig"(index := 25,
                           referenceDesignator := WSTRING#'BA030AZSDR26',
                           axisDB := "BA040AZSCDR26_MendrelAnodeRearAxisZ",
                           sinaType := "LAF_DRV_DIAG_SINA_TYPE_S120",
                           sinaHwID := "BA040AZSCU6~PROFINET_interface~BA040AZSDR26_SIEMENS_telegr,,,_2",
                           sinaDriveObjectNo := 5,
                           configuration := "DriveDiagConfig".driveObjects,
                           error => #tempError,
                           status => #tempStatus,
                           diagnostics => #tempDiagnostics);
   "LAF_SetDriveObjectConfig"(index := 26,
                           referenceDesignator := WSTRING#'BA030AZSDR27',
                           axisDB := "BA040AZSCDR27_MendrelCathodeFrontAxisY",
                           sinaType := "LAF_DRV_DIAG_SINA_TYPE_S120",
                           sinaHwID := "BA040AZSCU7~PROFINET_interface~BA040AZSDR27_SIEMENS_telegr,,,",
                           sinaDriveObjectNo := 5,
                           configuration := "DriveDiagConfig".driveObjects,
                           error => #tempError,
                           status => #tempStatus,
                           diagnostics => #tempDiagnostics);
   "LAF_SetDriveObjectConfig"(index := 27,
                           referenceDesignator := WSTRING#'BA030AZSDR28',
                           axisDB := "BA040AZSCDR28_MendrelCathodeFrontAxisZ",
                           sinaType := "LAF_DRV_DIAG_SINA_TYPE_S120",
                           sinaHwID := "BA040AZSCU7~PROFINET_interface~BA040AZSDR28_SIEMENS_telegr,,,",
                           sinaDriveObjectNo := 5,
                           configuration := "DriveDiagConfig".driveObjects,
                           error => #tempError,
                           status => #tempStatus,
                           diagnostics => #tempDiagnostics);
   "LAF_SetDriveObjectConfig"(index := 28,
                           referenceDesignator := WSTRING#'BA030AZSDR29',
                           axisDB := "BA040AZSCDR29_MendrelCathodeRearAxisY",
                           sinaType := "LAF_DRV_DIAG_SINA_TYPE_S120",
                           sinaHwID := "BA040AZSCU7~PROFINET_interface~BA040AZSDR29_SIEMENS_telegr,,,",
                           sinaDriveObjectNo := 5,
                           configuration := "DriveDiagConfig".driveObjects,
                           error => #tempError,
                           status => #tempStatus,
                           diagnostics => #tempDiagnostics);
   "LAF_SetDriveObjectConfig"(index := 29,
                           referenceDesignator := WSTRING#'BA030AZSDR30',
                           axisDB := "BA040AZSCDR30_MendrelCathodeRearAxisZ",
                           sinaType := "LAF_DRV_DIAG_SINA_TYPE_S120",
                           sinaHwID := "BA040AZSCU7~PROFINET_interface~BA040AZSDR30_SIEMENS_telegr,,,",
                           sinaDriveObjectNo := 5,
                           configuration := "DriveDiagConfig".driveObjects,
                           error => #tempError,
                           status => #tempStatus,
                           diagnostics => #tempDiagnostics);
   "LAF_SetDriveObjectConfig"(index := 30,
                           referenceDesignator := WSTRING#'BA030AZSDR31',
                           axisDB := "BA040AZSCDR31_StackTableAxisZ",
                           sinaType := "LAF_DRV_DIAG_SINA_TYPE_S120",
                           sinaHwID := "BA040AZSCU5~PROFINET_interface~BA040AZSDR31_SIEMENS_telegr,,,",
                           sinaDriveObjectNo := 5,
                           configuration := "DriveDiagConfig".driveObjects,
                           error => #tempError,
                           status => #tempStatus,
                           diagnostics => #tempDiagnostics);
   "LAF_SetDriveObjectConfig"(index := 31,
                           referenceDesignator := WSTRING#'BA030AZSDR32',
                           axisDB := "BA040AZSCDR32_StackTableOutFrontAxisZ",
                           sinaType := "LAF_DRV_DIAG_SINA_TYPE_S120",
                           sinaHwID := "BA040AZSCU5~PROFINET_interface~BA040AZSDR32_SIEMENS_telegr,,,",
                           sinaDriveObjectNo := 5,
                           configuration := "DriveDiagConfig".driveObjects,
                           error => #tempError,
                           status => #tempStatus,
                           diagnostics => #tempDiagnostics);
   "LAF_SetDriveObjectConfig"(index := 32,
                           referenceDesignator := WSTRING#'BA030AZSDR33',
                           axisDB := "BA040AZSCDR33_StackTableOutRearAxisZ",
                           sinaType := "LAF_DRV_DIAG_SINA_TYPE_S120",
                           sinaHwID := "BA040AZSCU5~PROFINET_interface~BA040AZSDR33_SIEMENS_telegr,,,",
                           sinaDriveObjectNo := 5,
                           configuration := "DriveDiagConfig".driveObjects,
                           error => #tempError,
                           status => #tempStatus,
                           diagnostics => #tempDiagnostics);
   "LAF_SetDriveObjectConfig"(index := 33,
                           referenceDesignator := WSTRING#'BA030AZSDR34',
                           axisDB := "BA040AZSCDR34_SepaClampnCutterAxisX",
                           sinaType := "LAF_DRV_DIAG_SINA_TYPE_S120",
                           sinaHwID := "BA040AZSCU8~PROFINET_interface~BA040AZSDR34_SIEMENS_telegr,,,",
                           sinaDriveObjectNo := 5,
                           configuration := "DriveDiagConfig".driveObjects,
                           error => #tempError,
                           status => #tempStatus,
                           diagnostics => #tempDiagnostics);
   "LAF_SetDriveObjectConfig"(index := 34,
                           referenceDesignator := WSTRING#'BA030AZSDR35',
                           axisDB := "BA040AZSCDR35_SepaClampnCutterAxisZ",
                           sinaType := "LAF_DRV_DIAG_SINA_TYPE_S120",
                           sinaHwID := "BA040AZSCU8~PROFINET_interface~BA040AZSDR35_SIEMENS_telegr,,,",
                           sinaDriveObjectNo := 5,
                           configuration := "DriveDiagConfig".driveObjects,
                           error => #tempError,
                           status => #tempStatus,
                           diagnostics => #tempDiagnostics);
   "LAF_SetDriveObjectConfig"(index := 35,
                           referenceDesignator := WSTRING#'BA030AZSDR36',
                           axisDB := "BA040AZSCDR36_SepaGripperAxisX",
                           sinaType := "LAF_DRV_DIAG_SINA_TYPE_S120",
                           sinaHwID := "BA040AZSCU8~PROFINET_interface~BA040AZSDR36_SIEMENS_telegr,,,",
                           sinaDriveObjectNo := 5,
                           configuration := "DriveDiagConfig".driveObjects,
                           error => #tempError,
                           status => #tempStatus,
                           diagnostics => #tempDiagnostics);
   "LAF_SetDriveObjectConfig"(index := 36,
                           referenceDesignator := WSTRING#'BA030AZSDR37',
                           axisDB := "BA040AZSCDR37_SepaGripperAxisZ",
                           sinaType := "LAF_DRV_DIAG_SINA_TYPE_S120",
                           sinaHwID := "BA040AZSCU8~PROFINET_interface~BA040AZSDR37_SIEMENS_telegr,,,",
                           sinaDriveObjectNo := 5,
                           configuration := "DriveDiagConfig".driveObjects,
                           error => #tempError,
                           status => #tempStatus,
                           diagnostics => #tempDiagnostics);
   "LAF_SetDriveObjectConfig"(index := 37,
                           referenceDesignator := WSTRING#'BA030AZSDR38',
                           axisDB := "BA040AZSCDR38_SepaGripperAxisC",
                           sinaType := "LAF_DRV_DIAG_SINA_TYPE_S120",
                           sinaHwID := "BA040AZSCU8~PROFINET_interface~BA040AZSDR38_SIEMENS_telegr,,,",
                           sinaDriveObjectNo := 5,
                           configuration := "DriveDiagConfig".driveObjects,
                           error => #tempError,
                           status => #tempStatus,
                           diagnostics => #tempDiagnostics);
   "LAF_SetDriveObjectConfig"(index := 38,
                           referenceDesignator := WSTRING#'BA030AZSDR39',
                           axisDB := "BA040AZSCDR39_JRWinderRearAxisY",
                           sinaType := "LAF_DRV_DIAG_SINA_TYPE_S120",
                           sinaHwID := "BA040AZSCU9~PROFINET_interface~BA040AZSDR39_SIEMENS_telegr,,,",
                           sinaDriveObjectNo := 5,
                           configuration := "DriveDiagConfig".driveObjects,
                           error => #tempError,
                           status => #tempStatus,
                           diagnostics => #tempDiagnostics);
   "LAF_SetDriveObjectConfig"(index := 39,
                           referenceDesignator := WSTRING#'BA030AZSDR40',
                           axisDB := "BA040AZSCDR40_JRWinderFrontAxisY",
                           sinaType := "LAF_DRV_DIAG_SINA_TYPE_S120",
                           sinaHwID := "BA040AZSCU9~PROFINET_interface~BA040AZSDR40_SIEMENS_telegr,,,",
                           sinaDriveObjectNo := 5,
                           configuration := "DriveDiagConfig".driveObjects,
                           error => #tempError,
                           status => #tempStatus,
                           diagnostics => #tempDiagnostics);
   "LAF_SetDriveObjectConfig"(index := 40,
                           referenceDesignator := WSTRING#'BA030AZSDR41',
                           axisDB := "BA040AZSCDR41_JRWinderAxisB",
                           sinaType := "LAF_DRV_DIAG_SINA_TYPE_S120",
                           sinaHwID := "BA040AZSCU8~PROFINET_interface~BA040AZSDR41_SIEMENS_telegr,,,",
                           sinaDriveObjectNo := 5,
                           configuration := "DriveDiagConfig".driveObjects,
                           error => #tempError,
                           status => #tempStatus,
                           diagnostics => #tempDiagnostics);
END_REGION

REGION Network 5: Manual Operation Line
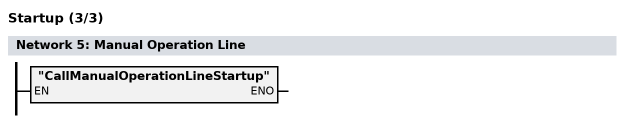
   RUNG wire#powerrail
      "CallManualOperationLineStartup"()
   END_RUNG
   // the same network as SCL:
   "CallManualOperationLineStartup"();
END_REGION
END_ORGANIZATION_BLOCK
